Universal Robots PolyScope program: extcontrol.urp

Program extcontrol (installation=default directory=/home/main/ursim-5.2.0.61336/programs createdIn=5.2.0.61336 lastSavedIn=5.2.0.61336 robotSerialNumber=20183599999)
Calibrated DH parameters: a=[0, -0.425, -0.3922, 0, 0, 0]; d=[0.1625, 0, 0, 0.1333, 0.0997, 0.0996]; alpha=[1.570796, 0, 0, 1.570796, -1.570796, 0]; deltaTheta=[0, 0, 0, 0, 0, 0]
Robot Program (runOnlyOnce=false)
  URCap External Control (External Control, FZI Research Center for Information Technology)
